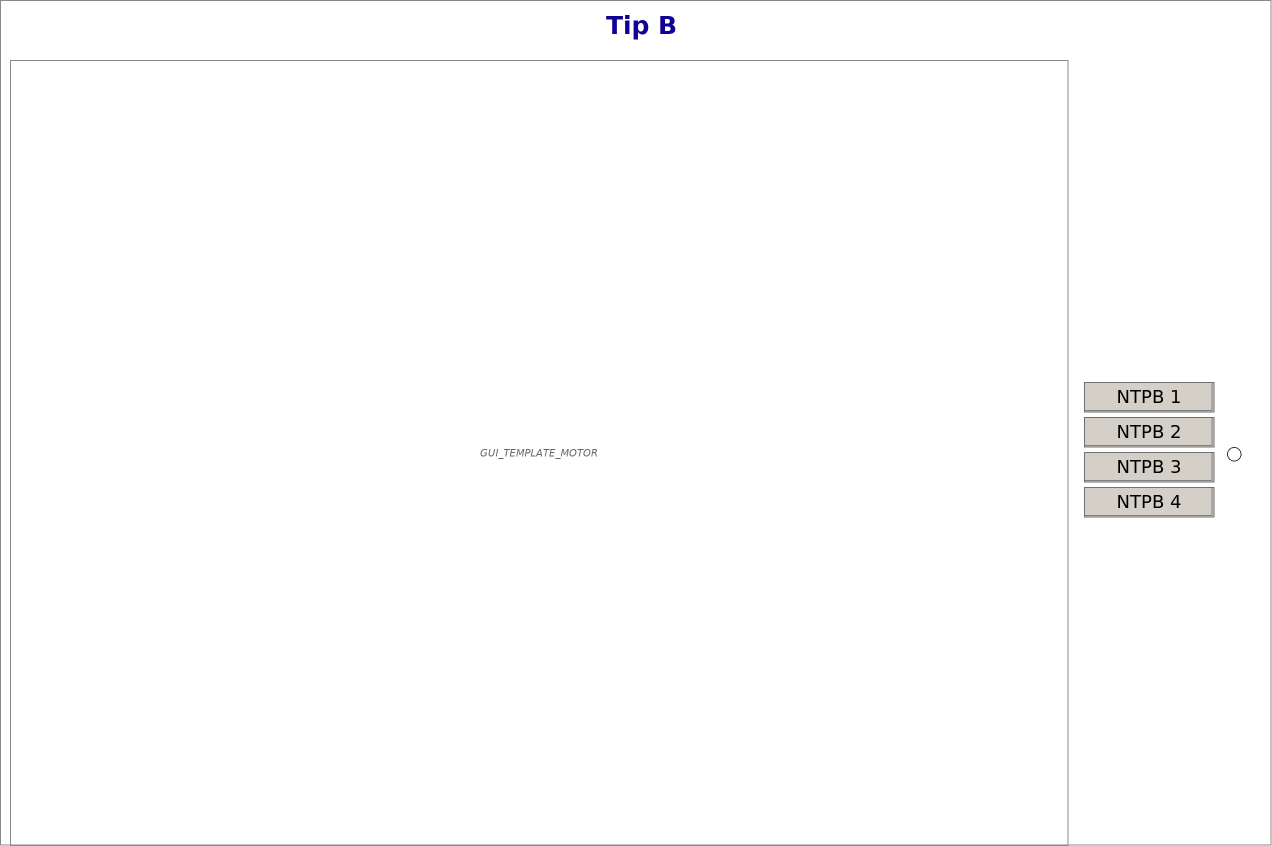
VISUALIZATION VISU_HMI_TIP_B  // 1272x846
    Label (542,10 199x30), "Tip B"
    Group (10,60 1262x786)
        Frame (0,0 1058x786)
            shows GUI_TEMPLATE_MOTOR(m_Instance := MAIN.nott_ics.TipTilt.ptrTipActuatorsB[MAIN.nott_ics.TipTilt.guiTipActuatorsBIndex]^)
        Group (1074,322 188x142)
            RadioButton (141,2 47x140), variable: MAIN.nott_ics.TipTilt.guiTipActuatorsBIndex-1
                Areas[0]: Text=Radiobutton
                Areas[1]: Text=Radiobutton
            Button (0,0 130x30), "NTPB 1"
                OnMouseClick: execute { MAIN.nott_ics.TipTilt.guiTipActuatorsBIndex := 1; }
            Button (0,35 130x30), "NTPB 2"
                OnMouseClick: execute { MAIN.nott_ics.TipTilt.guiTipActuatorsBIndex := 2; }
            Button (0,70 130x30), "NTPB 3"
                OnMouseClick: execute { MAIN.nott_ics.TipTilt.guiTipActuatorsBIndex := 3; }
            Button (0,105 130x30), "NTPB 4"
                OnMouseClick: execute { MAIN.nott_ics.TipTilt.guiTipActuatorsBIndex := 4; }
END_VISUALIZATION

(* stored: Version 1.1.0.1, ProductVersion 3.1.4024.14
   Visu VISU_HMI_TIP_B: Id {7e4bb0ee-a0e5-47c2-8dd5-ac16ade33419} *)
